{attribute 'qualified_only'}
{attribute 'strict'}
{attribute 'to string'}
TYPE E_EventType :
(
	Alarm,
	Message
);
END_TYPE

(* stored: Version 1.1.0.1, ProductVersion 3.1.4024.11
   DUT E_EventType: Id {935007b8-6511-4731-a032-e2a2b1839aa4} *)
